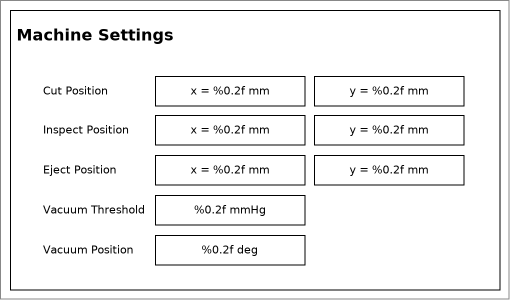
VISUALIZATION Settings_Mandrel  // 510x300
VAR_IN_OUT
	CutPositionX	: LREAL;
	CutPositionY	: LREAL;
	InspectPositionX: LREAL;
	InspectPositionY: LREAL;
	EjectPositionX	: LREAL;
	EjectPositionY	: LREAL;
	VacuumThreshold	: REAL;
	VacuumPosition : LREAL;
END_VAR
    Rectangle (10,10 490x280)
    Label (20,20 150x30), "Machine Settings"
    Label (40,76 90x30), "Cut Position"
    Label (40,115 90x30), "Inspect Position"
    Label (40,155 90x30), "Eject Position"
    Rectangle (155,76 150x30), "x = %0.2f mm", text variable: CutPositionX
        OnMouseClick: write CutPositionX via Default
    Rectangle (314,76 150x30), "y = %0.2f mm", text variable: CutPositionY
        OnMouseClick: write CutPositionY via Default
    Rectangle (155,115 150x30), "x = %0.2f mm", text variable: InspectPositionX
        OnMouseClick: write InspectPositionX via Default
    Rectangle (314,115 150x30), "y = %0.2f mm", text variable: InspectPositionY
        OnMouseClick: write InspectPositionY via Default
    Rectangle (155,155 150x30), "x = %0.2f mm", text variable: EjectPositionX
        OnMouseClick: write EjectPositionX via Default
    Rectangle (314,155 150x30), "y = %0.2f mm", text variable: EjectPositionY
        OnMouseClick: write EjectPositionY via Default
    Label (40,195 110x30), "Vacuum Threshold"
    Rectangle (155,195 150x30), "%0.2f mmHg", text variable: VacuumThreshold
        OnMouseClick: write VacuumThreshold via Default
    Label (40,235 110x30), "Vacuum Position"
    Rectangle (155,235 150x30), "%0.2f deg", text variable: VacuumPosition
        OnMouseClick: write VacuumPosition via Default, min 0, max 13000, title 'Vacuum Axis Position'
END_VISUALIZATION

(* stored: Version 1.1.0.1, ProductVersion 3.1.4024.9
   Visu Settings_Mandrel: Id {9fb065b9-6319-4a88-8b94-9e707f6c33bb} *)
